PROGRAM MAIN
VAR
  mathTest : MathTest;
  minDurationTest : MinDurationTest;
  velocityInterfaceTest : VelocityInterfaceTest;
  knownExamplesTest : KnownExamplesTest;
  secondaryFeaturesTest : SecondaryFeaturesTest;
  debuggedExamplesTest : DebuggedExamplesTest;
  targetPosTest : TargetPosTest;
  targetPosAccTest : TargetPosAccTest;
  targetPosVelTest : TargetPosVelTest;
  targetPosVelAccTest : TargetPosVelAccTest;
  propagateTest : PropagateTest;
  // generatedTest : GeneratedTest;
END_VAR

TcUnit.RUN();

END_PROGRAM

(* stored: Version 1.1.0.1, ProductVersion 3.1.4024.9
   POU MAIN: Id {f725f308-f3c1-4da3-8197-2078a75fc02b}, SpecialFunc None *)
